// TIA Portal V19 export
TYPE "LEXCHANGETRAY_typeRoller_interface_B2"
// stored: Access Published
   STRUCT
      init : Bool;
      deliver : "LEXCHANGETRAY_typeRoller_deliver_interface_B2";
      recieve : "LEXCHANGETRAY_typeRoller_recieve_interface_B2";
   END_STRUCT;
END_TYPE
